Fanuc KAREL source: MP0297.KL

-- PROVISIONAL review KL for V1013-1; original PC SHA256 bbe6d4f487ecdd8accffdebda4e1b75d08cc16d02b0ddce323ccecf00e5efb4c
-- Incomplete behavior may be omitted. Consult companion uncertainty JSON. Do not deploy.
PROGRAM MP0297
%NOLOCKGROUP
-- UNRESOLVED_LOCAL_POOL 8 cells at code offset 61; source declarations unknown
-- DIRECT_LOCAL_WORD_ACCESS alone does not prove INTEGER, REAL, or BOOLEAN
BEGIN
  -- UNRESOLVED_PC offsets 0-1; opcodes 7B
  -- UNRESOLVED_PC offsets 6-18; opcodes 2D,9D,52,7F
  -- UNRESOLVED_PC offsets 23-28; opcodes 7F,7B
  -- UNRESOLVED_PC offsets 33-49; opcodes 2D,2E,69,7F
  -- UNRESOLVED_PC offsets 54-66; opcodes 7F,2B,2C,7B
  -- UNRESOLVED_PC offsets 71-82; opcodes 2E,23
  -- UNRESOLVED_PC offsets 87-98; opcodes 2E,23
  -- UNRESOLVED_PC offsets 103-114; opcodes 2E,23
  -- UNRESOLVED_PC offsets 119-130; opcodes 2E,23
  -- UNRESOLVED_PC offsets 135-146; opcodes 2E,23
  -- UNRESOLVED_PC offsets 151-162; opcodes 2E,23
  -- UNRESOLVED_PC offsets 167-185; opcodes 2E,21,69,23
  -- UNRESOLVED_PC offsets 190-194; opcodes 7F
  -- UNRESOLVED_PC offsets 199-215; opcodes 27,27,2E,27,2E,AA
  -- UNRESOLVED_PC offsets 220-224; opcodes 7F
END MP0297
